	16#4417: sMsg := '4417 parameter „Tolerance window for modulo-start” The value for the tolerance window for the modulo-axis-start is invalid. The value must be greater or equal than zero and smaller than the half encoder modulo-perio…';
	16#4418: sMsg := '4418 parameter „Encoder reference mode” The value for the encoder reference mode is not allowed, resp. is not supported for this encoder type.';
	16#4419: sMsg := '4419 parameter „Encoder evaluation direction” The value for the encoder evaluation direction (log. counter direction) is not allowed.';
	16#441A: sMsg := '441A parameter „Encoder reference system” The value for the encoder reference system is invalid (0: incremental, 1: absolute, 2: absolute+modulo).';
	16#441B: sMsg := '441B parameter „Encoder position initialization mode” When starting the TC system the value for the encoder position initialization mode is invalid.';
	16#441C: sMsg := '441C parameter „Encoder sign interpretation (UNSIGNED- / SIGNED- data type)” The value for the encoder sign interpretation (data type) for the encoder the actual increment calculation (0: Default/not defined, 1: UNS…';
	16#4420: sMsg := '4420 parameter "Software end location monitoring minimum not allowed" The value for the activation of the software location monitoring minimum is not allowed.';
	16#4421: sMsg := '4421 parameter "Software end location monitoring maximum not allowed" The value for the activation of the software location monitoring maximum is not allowed.';
	16#4422: sMsg := '4422 function "Actual value setting is outside the value range" The "set actual value" function cannot be carried out, because the new actual position is outside the expected range of values.';
	16#4423: sMsg := '4423 parameter "Software end location minimum not allowed" The value for the software end location minimum is not allowed.';
	16#4424: sMsg := '4424 parameter "Software end location maximum not allowed" The value for the software end location maximum is not allowed.';
	16#4425: sMsg := '4425 parameter „Filter mask for the raw data of the encoder is invalid” The value for the filter mask of the encoder raw data in increments is invalid.';
	16#4426: sMsg := '4426 parameter „Reference mask for the raw data of the encoder is invalid” The value for the reference mask (increments per encoder turn, absolute resolution) for the raw data of the encoder is invalid. E.g. this va…';
	16#4430: sMsg := '4430 function "Hardware latch activation (encoder)" Activation of the encoder hardware latch was implicitly initiated by the referencing procedure. If this function has already been activated but a latch value has …';
	16#4431: sMsg := '4431 function "External hardware latch activation (encoder)" The activation of the external hardware latch (only available on the KL5101) is initiated explicitly by an ADS command (called from the PLC program of th…';
	16#4432: sMsg := '4432 function "External hardware latch activation (encoder)" If a referencing procedure has previously been initiated and the hardware still signals a valid latch value ("latch valid"), this function must not be ca…';
	16#4433: sMsg := '4433 function "External hardware latch activation (encoder)" If this function has already been initiated and the hardware is still signaling that the external latch value is still valid ("extern latch valid"), a fu…';
	16#4434: sMsg := '4434 monitoring "Encoder function not supported" An encoder function has been activated that is currently not released for use, or which is not even implemented.';
	16#4435: sMsg := '4435 monitoring „Encoder function is already active” An encoder function can not been activated because this functionality is already active.';
	16#4440: sMsg := '4440 initialization "Encoder initialization" Encoder has not been initialized. Although the axis has been created, the rest of the initialization has not been performed (1. Initialization of axis I/O, 2. Initialization o…';
	16#4441: sMsg := '4441 address "Axis address" The encoder does not have an axis, or the axis address has not been initialized.';
	16#4442: sMsg := '4442 address "I/O input structure address" The drive does not have a valid I/O input address in the process image.';
	16#4443: sMsg := '4443 address "I/O output structure address" The encoder does not have a valid I/O output address in the process image.';
	16#4450: sMsg := '4450 monitoring "Encoder counter underflow monitoring" The encoders incremental counter has underflowed.';
	16#4451: sMsg := '4451 monitoring "Encoder counter overflow monitoring" The encoders incremental counter has overflowed.';
	16#4460: sMsg := '4460 monitoring "Software end location minimum (axis start)" With active monitoring of the software end location for a minimum, a start has been made from a position that lies below the software end location minimum.…';
	16#4461: sMsg := '4461 monitoring "Software end location maximum (axis start)" With active monitoring of the software end location for a maximum, a start has been made from a position that lies above the software end location maximum.…';
	16#4462: sMsg := '4462 monitoring "Software end location minimum (positioning process)" With active monitoring of the software end location for a minimum, the actual position has fallen below the software end location minimum. In the …';
	16#4463: sMsg := '4463 monitoring "Software end location maximum (positioning process)" With active monitoring of the software end location for a maximum, the actual position has exceeded the software end location maximum. In the case…';
	16#4464: sMsg := '4464 monitoring „Encoder hardware error” The drive resp. the encoder system reports a hardware error of the encoder. An optimal error code is displayed in the message of the event log.';
	16#4465: sMsg := '4465 monitoring „Position initialization error at system start” At the first initialization of the set position was this for all initialization trials (without over-/under-flow, with underflow and overflow ) out of t…';
	16#4470: sMsg := '4470 monitoring "SSI transformation fault or not finished" The SSI transformation of the FOX 50 module was faulty for some NC-cycles or did not finished respectively.';
	16#44A2: sMsg := '44A2 monitoring "ENCERR_ADDR_CONTROLLER"';
	16#44A3: sMsg := '44A3 monitoring "ENCERR_INVALID_CONTROLLERTYPE"';
	16#4500: sMsg := '4500 parameter "Controller ID not allowed" The value for the controller ID is not allowed, e.g. because it has already been assigned, is less than or equal to zero, or is greater than 255.';
	16#4501: sMsg := '4501 parameter "Controller type not allowed" The value for the controller type is unacceptable because it is not defined. Type 1: P-controller (position) . . . Type 7: High/low speed controller Type 8: Stepper motor…';
	16#4502: sMsg := '4502 parameter "Controller operating mode not allowed" The value for the controller operating mode is not allowed.';
	16#4503: sMsg := '4503 parameter "Weighting of the velocity pre-control not allowed" The value for the percentage weighting of the velocity pre-control is not allowed. The parameter is pre-set to 1.0 (100%) as standard.';
	16#4504: sMsg := '4504 parameter "Following error monitoring (position) not allowed" The value for the activation of the following error monitoring is not allowed.';
	16#4505: sMsg := '4505 parameter "Following error (velocity) not allowed" The value for the activation of the following error monitoring (velocity) is not allowed.';
	16#4506: sMsg := '4506 parameter "Following error window (position) not allowed" The value for the following error window (maximum allowable following error) is not allowed.';
	16#4507: sMsg := '4507 parameter "Following error filter time (position) not allowed" The value for the following error filter time (position) is not allowed.';
	16#4508: sMsg := '4508 parameter "Following error window (velocity) not allowed" The value for the following error window (velocity) is not allowed.';
	16#4509: sMsg := '4509 parameter "Following error filter time (velocity) not allowed" The value for the following error filter time (velocity) is not allowed.';
	16#4510: sMsg := '4510 parameter "Proportional gain Kv or Kp (position controller) not allowed" The value for the proportional gain (Kv factor or Kp factor) is not allowed.';
	16#4511: sMsg := '4511 parameter "Integral-action time Tn (position controller) not allowed" The value for the integral-action time is not allowed (I proportion of the PID T1 controller).';
	16#4512: sMsg := '4512 parameter "Derivative action time Tv (position controller) not allowed" The value for the derivative action time is not allowed (D proportion of the PID T1 controller).';
	16#4513: sMsg := '4513 parameter "Damping time Td (position controller) not allowed" The value for the damping time is not allowed (D proportion of the PID T1 controller). Suggested value: 0.1 * Tv';
	16#4514: sMsg := '4514 function "Activation of the automatic offset compensation not allowed" Activation of the automatic offset compensation is only possible for certain types of controller (with no I component).';
	16#4515: sMsg := '4515 parameter "Additional proportional gain Kv or Kp (position controller) not allowed" The value for the second term of the proportional gain (Kv factor or Kp factor) is not allowed.';
	16#4516: sMsg := '4516 parameter "Reference velocity for additional proportional gain Kv or Kp (position controller) not allowed" The value for the reference velocity percentage data entry, to which the additional proportional gain i…';
	16#4517: sMsg := '4517 parameter "Proportional gain Pa (acceleration proportion) not allowed" The value for the proportional gain (Pa factor) is not allowed.';
	16#4518: sMsg := '4518 parameter "Proportional gain Kv (velocity controller) not allowed" The value for the proportional gain (Kv factor) is not allowed.';
	16#4519: sMsg := '4519 parameter “Reset time Tn (velocity controller) not allowed” The value for the integral-action time is not allowed (I proportion of the PID T1 controller).';
	16#451A: sMsg := '451A address "CONTROLERR_RANGE_ACCJUMPLIMITINGMODE"';
	16#451B: sMsg := '451B address "CONTROLERR_RANGE_ACCJUMPVALUE"';
	16#451C: sMsg := '451C address "CONTROLERR_RANGE_FILTERTIME"';
	16#451D: sMsg := '451D parameter „Dead zone not allowed” The value for the dead zone from the position error or the velocity error (system deviation) is not allowed (only for complex controller with velocity or torque interface).';
	16#4520: sMsg := '4520 parameter ”Rate time Tv (velocity controller) not allowed” The value for the derivative action time is not allowed (D proportion of the PID T1 controller).';
	16#4521: sMsg := '4521 parameter "Damping time Td (velocity controller) not allowed" The value for the damping time is not allowed (D proportion of the PID T1 controller). Suggested value: 0.1 * Tv';
	16#4522: sMsg := '4522 parameter "CONTROLERR_RANGE_IOUTPUTLIMIT"';
	16#4523: sMsg := '4523 parameter "CONTROLERR_RANGE_DOUTPUTLIMIT"';
	16#4524: sMsg := '4524 parameter "CONTROLERR_RANGE_POSIDISABLEWHENMOVING"';
	16#4540: sMsg := '4540 initialization "Controller initialisation" Controller has not been initialised. Although the controller has been created, the rest of the initialisation has not been performed (1. Initialisation of controller, 2. Re…';
	16#4541: sMsg := '4541 address "Axis address" Controller does not know its axis, or the axis address has not been initialised.';
	16#4542: sMsg := '4542 address "Drive address" Controller does not know its drive, or the drive address has not been initialised.';
	16#4550: sMsg := '4550 monitoring "Following error monitoring (position)" With active following error monitoring (position) a following error exceedance has occurred, whose magnitude is greater than the following error window, and who…';
	16#4551: sMsg := '4551 monitoring "Following error monitoring (velocity)" With active following error monitoring (velocity) a velocity following error exceedance has occurred, whose magnitude is greater than the following error window…';
	16#45A0: sMsg := '45A0 monitoring "CONTROLERR_RANGE_AREA_ASIDE"';
	16#45A1: sMsg := '45A1 monitoring "CONTROLERR_RANGE_AREA_BSIDE"';
	16#45A2: sMsg := '45A2 monitoring "CONTROLERR_RANGE_QNENN"';
	16#45A3: sMsg := '45A3 monitoring "CONTROLERR_RANGE_PNENN"';
	16#45A4: sMsg := '45A4 monitoring "CONTROLERR_RANGE_AXISIDPRESP0"';
	16#4600: sMsg := '4600 parameter "Drive ID not allowed" The value for the drive ID is not allowed, e.g. because it has already been assigned, is less than or equal to zero, or is greater than 255.';
	16#4601: sMsg := '4601 parameter "Drive type not allowed" The value for the drive type is unacceptable because it is not defined.';
	16#4602: sMsg := '4602 parameter "Drive operating mode not allowed" The value for the drive operating mode is not allowed. Modus 1: Standard';
	16#4603: sMsg := '4603 parameter "Motor polarity inverted?" The flag for the motor polarity is not allowed. Flag 0: Positive motor polarity Flag 1: Negative motor polarity';
	16#4604: sMsg := '4604 parameter "Drift compensation/velocity offset (DAC offset)" The value for the drift compensation (DAC offset) is not allowed.';
	16#4605: sMsg := '4605 parameter "Reference velocity (velocity pre-control)" The value for the reference velocity (velocity pre-control) is not allowed.';
	16#4606: sMsg := '4606 parameter "Reference output in percent" The value for the reference output in percent is not allowed. The value 1.0 (100 %) usually corresponds to a voltage of 10.0 V.';
	16#4607: sMsg := '4607 parameter "Quadrant compensation factor" The value for the quadrant compensation factor is not allowed.';
	16#4608: sMsg := '4608 parameter "Velocity reference point in percent" The value for the velocity reference point in percent is not allowed. The value 1.0 corresponds to 100 percent.';
	16#4609: sMsg := '4609 parameter "Output reference point in percent" The value for the output reference point in percent is not allowed. The value 1.0 corresponds to 100 percent.';
	16#460A: sMsg := '460A parameter "Minimum or maximum output limit" The values for the minimum and/or maximum output limit is not allowed. This will happen if the range of values is exceeded, the maximum limit is smaller than the mini…';
	16#460B: sMsg := '460B parameter "DRIVEERR_RANGE_MAXINCREMENT"';
	16#460C: sMsg := '460C parameter "DRIVEERR_RANGE_ DRIVECONTROLDWORD"';
	16#460D: sMsg := '460D parameter "DRIVEERR_RANGE_ RESETCYCLECOUNTER"';
	16#460F: sMsg := '460F parameter „Drive torque output scaling is not allowed” The value for the drive torque output scaling (rotary motor) or the force output scaling (linear motor) is not allowed.';
	16#4610: sMsg := '4610 parameter „Drive velocity output scaling is not allowed” The value for the drive velocity output scaling is not allowed.';
	16#4611: sMsg := '4611 parameter "Profi Drive DSC Proportional gain Kpc (position controller) not allowed" The value for the profi drive DSC proportional gain (Kpc factor) is not allowed.';
	16#4612: sMsg := '4612 parameter „Table-ID is invalid” The value for the table-ID is invalid.';
	16#4613: sMsg := '4613 parameter „Table interpolationtype is invalid” The value for the table interpolation-type is invalid.';
	16#4614: sMsg := '4614 parameter „Outputoffset in percent is invalid” The value for the output offset in percent (+/- 1.0) is invalid.';
	16#4615: sMsg := '4615 parameter „Profi Drive DSC scaling factor for calculating Xerr (position controller) is not allowed” The value as profi drive DSC scaling factor for calculating Xerr is invalid.';
	16#4616: sMsg := '4616 parameter „Drive acceleration output scaling is not allowed” The value for the drive acceleration/deceleration output scaling is not allowed.';
	16#4617: sMsg := '4617 parameter „Drive position output scaling is not allowed” The value for the drive position output scaling is not allowed.';
	16#4620: sMsg := '4620 parameter "Bit mask for stepper motor cycle not allowed" A value in the various stepper motor masks for the cycle concerned is not allowed.';
	16#4621: sMsg := '4621 parameter "Bit mask for stepper motor holding current not allowed" The value for the stepper motor holding mask is not allowed.';
	16#4630: sMsg := '4630 monitoring „Overtemperature” The drive resp. terminal detects an overtemperature alarm.';
	16#4631: sMsg := '4631 monitoring „Undervoltage” The drive resp. terminal detects an undervoltage (supply voltage to low).';
	16#4632: sMsg := '4632 monitoring „Wire breakage in phase A” The drive resp. terminal detects a wire breakage in phase A.';
	16#4633: sMsg := '4633 monitoring „Wire breakage in phase B” The drive resp. terminal detects a wire breakage in phase B.';
	16#4634: sMsg := '4634 monitoring „Overcurrent in phase A” The drive resp. terminal detects an overcurrent in phase A.';
	16#4635: sMsg := '4635 monitoring „Overcurrent in Phase B” The drive resp. terminal detects an overcurrent in phase B.';
	16#4636: sMsg := '4636 monitoring „Torque overload (stall situation)” The drive resp. terminal detects a torque overload (stall situation).';
	16#4640: sMsg := '4640 initialization "Drive initialisation" Drive has not been initialised. Although the drive has been created, the rest of the initialisation has not been performed (1. Initialisation of drive I/O, 2. Initialisation of …';
	16#4641: sMsg := '4641 address "Axis address" Drive does not know its axis, or the axis address has not been initialised.';
	16#4642: sMsg := '4642 address "I/O input structure address" The drive does not have a valid I/O input address in the process image.';
	16#4643: sMsg := '4643 address "I/O output structure address" The drive does not have a valid I/O output address in the process image.';
	16#4650: sMsg := '4650 monitoring "Drive not ready for operation" The drive is not ready for operation. The following are possible causes: - the drive is in failure state (hardware fault) - the drive is in the starting-up stage…';
	16#4651: sMsg := '4651 monitoring "Error in cyclic communication with the drive (life counter)"';
	16#4652: sMsg := '4652 monitoring "Not permitted to change the table ID while the axis is enabled"';
	16#4655: sMsg := '4655 monitoring "Invalid IO data for more than n consecutive nc cycles"';
	16#4A00: sMsg := '4A00 parameter "Table ID not allowed" The value for the table ID is not allowed, e.g. because it has already been assigned, is less than or equal to zero, or is greater than 255.';
	16#4A01: sMsg := '4A01 parameter "Table type not allowed" The value for the table type is unacceptable because it is not defined.';
	16#4A02: sMsg := '4A02 parameter "Number of lines in the table not allowed" The value of the number of lines in the table is not allowed, because, for example, it is smaller than two at linear interpolation and smaller than four at s…';
	16#4A03: sMsg := '4A03 parameter "Number of columns in the table is not allowed" The value of the number of columns in the table is not allowed, because, for example, it is less than or equal to zero (depends upon the type of table o…';
	16#4A04: sMsg := '4A04 parameter "Step size (position delta) not allowed" The value for the step size between two lines (position delta) is not allowed, because, for example, it is less than or equal to zero.';
	16#4A05: sMsg := '4A05 parameter "Period not allowed" The value for the period is not allowed, because, for example, it is less than or equal to zero.';
	16#4A06: sMsg := '4A06 parameter "Table is not monotonic" The value for the step size is not allowed, because, for example, it is less than or equal to zero.';
	16#4A07: sMsg := '4A07 initialization „Table sub type is not allowed” The value for the table sub type is not allowed or otherwise the table class (slave type) do not match up to the table main type.';
	16#4A08: sMsg := '4A08 initialization „Table interpolation type is not allowed” The value for the table interpolation type is allowed.';
	16#4A09: sMsg := '4A09 initialization "Incorrect table main type" The table main type is unknown or otherwise the table class (slave type) do not match up to the table main type.';
	16#4A10: sMsg := '4A10 initialization "Table initialisation" Table has not been initialised. Although the table has been created, the rest of the initialisation has not been performed. For instance, the number of lines or columns may be l…';
	16#4A11: sMsg := '4A11 initialization "Not enough memory" Table could not be created, since there is not enough memory.';
	16#4A12: sMsg := '4A12 function "Function not executed, function not available" The function has not been implemented, or cannot be executed, for the present type of table.';
	16#4A13: sMsg := '4A13 function "Line index not allowed" The start line index or the stop line index to be used for read or write access to the table is not allowed. For instance, the line index may be greater than the total number …';
	16#4A14: sMsg := '4A14 function "Column index not allowed" The start column index or the stop column index to be used for read or write access to the table in not allowed. For instance, the column index may be greater than the total…';
	16#4A15: sMsg := '4A15 function "Number of lines not allowed" The number of lines to be read from or written to the table is not allowed. The number of lines must be an integer multiple of the number of elements in a line (n * numbe…';
	16#4A16: sMsg := '4A16 function "Number of columns not allowed" The number of columns to be read from or written to the table is not allowed. The number of columns must be an integer multiple of the number of elements in a column (n…';
	16#4A17: sMsg := '4A17 function "Error in scaling or in range entry" The entries in the table header are inconsistent, e.g. the validity range is empty. If the error is generated during the run time it is a run time error and stops …';
	16#4A18: sMsg := '4A18 function "Multi table slave out of range" The slave master position is outside the table values for the master. The error is a run-time error, and stops the master/slave group.';
	16#4A19: sMsg := '4A19 function "Solo table underflow" The slave master position is outside the table values for the master. The master value of the equidistant table, to be processed linearly, lies under the first table value. The …';
	16#4A1A: sMsg := '4A1A function "Solo table overflow" The slave master position is outside the table values for the master. The master value of the equidistant table, to be processed linearly, lies above the first table value. The e…';
	16#4A1B: sMsg := '4A1B parameter "Incorrect execution mode" The cyclic execution mode can only be "true" or "false".';
	16#4A1C: sMsg := '4A1C parameter "Impermissible parameter" The Fifo parameter is not allowed.';
	16#4A1D: sMsg := '4A1D parameter "Fifo is empty" The Fifo of the external generator is empty. This can signify end of track or a run time error.';
	16#4A1E: sMsg := '4A1E parameter "Fifo is full" The Fifo of the external generator is full. It is the user‘s task to continue to attempt to fill the Fifo with the rejected values.';
	16#4A1F: sMsg := '4A1F parameter „Point-Index of Motion Function invalid” The point index of a Motion Function Point of a Function Table is invalid. First the point index has to be larger than zero and second it has to be numerical c…';
	16#4A20: sMsg := '4A20 initialization „No diagonalisation of matrix” The spline can not be calculated. The master positions are not correct.';
	16#4A21: sMsg := '4A21 initialization „Number of spline points to less” The number of points of a cubic spline has to be greater than two.';
	16#4A22: sMsg := '4A22 initialization „Fifo must not be overwritten” Fifo must not be overwritten since then the active line would be overwritten. It is the task of the user to secure that the active line is not modified.';
	16#4B00: sMsg := '4B00 parameter "Axis has been stopped" The axis has been stopped while the axis moves to target position. The axis could be stopped with a PLC Command via ADS, with the call of AXFNC or with the TwinCAT System Manag…';
	16#4B01: sMsg := '4B01 parameter "Axis cannot be started" The axis cannot be started, because:';
	16#4B02: sMsg := '4B02 parameter "Control mode not allowed" No Target Position Control and no Position Area Control.';
	16#4B03: sMsg := '4B03 parameter "Axis is not moving" Restart position and velocity is only allowed if axis is physically moving.';
	16#4B04: sMsg := '4B04 parameter "Wrong mode for RestartPosAndVelo" Wrong mode.';
	16#4B05: sMsg := '4B05 parameter "Command not allowed"';
	16#4B06: sMsg := '4B06 parameter "Parameter not correct"';
	16#4B07: sMsg := '4B07 parameter "Timeout axis function block"';
	16#4B08: sMsg := '4B08 parameter "Axis in protected mode" Axis is in protected mode (i.e. coupled) and cannot be moved.';
	16#4B09: sMsg := '4B09 parameter "Axis is not ready" Axis is not ready and cannot be moved.';
	16#4B0A: sMsg := '4B0A parameter "Homing error" The Homing of an axis could not be started or was not successful';
	16#4B0B: sMsg := '4B0B parameter "Invalid definition trigger input definition" The definition of the trigger signal used with the function block MC_TouchProbe is invalid. The defined encoder ID, the trigger signal or the trigger sign…';
	16#4B0C: sMsg := '4B0C function "position latch has been deactivated" The function block MC_TouchProbe encountered that a touch probe sequence has been deactivated after the block started this sequence. The reason for instance can b…';
	16#4B0D: sMsg := '4B0D function "Timeout NC status feedback" A function block has successfully executed a command but the NC does not pass the expected feedback in the axis status word.';
	16#4B0E: sMsg := '4B0E function "Supplement not installed" - The function is available as supplement product but not installed on the system.';
	16#4B0F: sMsg := '4B0F function "Timeout Register Access" - The access to a bus terminal register timed out.';
	16#4B10: sMsg := '4B10 function "M-Function request missing" This error occurs if a confirmation of an M-Function is made but the request bit is not set.';
	16#4B11: sMsg := '4B11 parameter "Zero shift index is out of range" The index of the zero shift is invalid';
	16#4B12: sMsg := '4B12 parameter "R parameter index or size is invalid". This error occurs, if the R parameters are written or read and the index or size is out of range';
	16#4B13: sMsg := '4B13 parameter "Index for tool description is invalid"';
	16#4B14: sMsg := '4B14 function "Version of cyclic channel interface does not match to the requested function and function block, resp." This error occurs, if an older TwinCAT Version is used and a new functionality from a newer TcN…';
	16#4B15: sMsg := '4B15 function "Channel is not ready for requested function". The requested function can not be executed due to a wrong state of the channel. This error occurs for instance, if retrace is requested and the axes are …';
	16#4B16: sMsg := '4B16 function "Requested function is not turned on". The requested function requires an explicit activation before it can be executed.';
	16#4B20: sMsg := '4B20 parameter "Cannot append all axes". This error occurs, if you want to append an auxiliary axes to an interpolation group and the function fails. Probably a prior assignment of an auxiliary axes was skipped.';
	16#4B30: sMsg := '4B30 parameter "Pointer invalid". The pointer to a data structure is invalid, e.g. NULL.';
	16#4B31: sMsg := '4B31 parameter "Size of memory invalid". The size parameter is invalid.';
	16#4B32: sMsg := '4B32 parameter "Invalid cam table ID". The cam table ID is out of the range from 1 to 255.';
	16#4B33: sMsg := '4B33 parameter "Invalid point ID". The point ID of a motion function point is lower than 1.';
	16#4B34: sMsg := '4B34 parameter "Invalid number of points ". The number of points to read or write is less than 1.';
	16#4B35: sMsg := '4B35 parameter "Invalid MC table type". The type of a cam table does not match the MC_TableType definition.';
	16#4B36: sMsg := '4B36 parameter "Invalid number of rows". The number of rows of a cam table is less than 1.';
	16#4B37: sMsg := '4B37 parameter "Invalid number of columns". The number of columns of a cam table is invalid.';
	16#4B38: sMsg := '4B38 parameter "Invalid Increment". The increment for an interpolation is invalid, e.g. <= 0.';
	16#4B40: sMsg := '4B40 monitoring "Unsupported Terminal Type". The terminal in use is not supported by this function block.';
	16#4B41: sMsg := '4B41 monitoring "Register Read/Write Error". This error implies to be a validation error.';
	16#4B42: sMsg := '4B42 monitoring "Axis is Enabled". Axis is enabled and is not supposed to be enabled for this operation';
	16#4B43: sMsg := '4B43 parameter "Size of compensation table wrong". The stated table size in bytes is not conform with the real size.';
	16#4B44: sMsg := '4B44 parameter The minimum/ maximum position of the compenstation table is not conform to the position in the table description (ST_CompensationDesc)';
	16#4B45: sMsg := '4B45 parameter "Not implemented". The requested function is not implemented in this combination.';
	16#4B60: sMsg := '4B60 monitoring "Motion command not be activated". A motion command has been started and has been buffered and confirmed by the NC. Nevertheless the command did not become active.';
	16#4B61: sMsg := '4B61 monitoring "Motion command could not be monitored by the PLC". A motion command has been started and has been buffered and confirmed by the NC. The PLC has not been able to monitor the execution of this command……';
	16#4B62: sMsg := '4B62 monitoring "Buffered command finished with error". A buffered command finished with an error. The error number is not available because a new command is already in execution.';
	16#4B63: sMsg := '4B63 monitoring "Buffered command finished without state feedback". A buffered command finished without success or error feedback.';
	16#4B64: sMsg := '4B64 monitoring "  BufferMode  not supported". The  BufferMode  is not supported by the command.';
	16#4B65: sMsg := '4B65 monitoring "Command number is zero". The system administrated command number for buffered commands is zero. ';
	16#4B71: sMsg := '4B71 parameter "Invalid NCI Entry Type". FB_NciFeedTablePreparation is called with an unknown nEntryType';
	16#4B72: sMsg := '4B72 function "NciFeedTable full". The table is full filled and therefore this entry is not accepted.';
	16#4B73: sMsg := '4B73 function internal error';
	16#4B74: sMsg := '4B74 parameter "ST_NciTangentialFollowingDesc: tangential axis is not an auxiliary axis" The entry ST_NciTangentialFollowingDesc contains an tangential axis that is no auxiliary axis.';
	16#4B75: sMsg := '4B75 parameter ST_NciTangentialFollowingDesc: nPathAxis1 and nPathAxis2, resp. are no path axes. So it is not possible to determine the plane.';
	16#4B76: sMsg := '4B76 parameter ST_NciTangentialFollwoingDesc: nPathAxis1 and nPathAxis2 are equal. So it is not possible to determine the plane.';
	16#4B77: sMsg := '4B77 parameter ST_NciGeoCirclePlane: circle is programmed in a wrong manner.';
	16#4B78: sMsg := '4B78 function Internal error in calculation of the tangential following';
	16#4B79: sMsg := '4B79 monitoring Tangential following: With ST_NciTangentialFollowingDesc the monitoring of the deviation angle (E_TfErrorOnCrirical1) is activated and with the actual segment the deviation angle is too big.';
	16#4B7A: sMsg := '4B7A function not implemented';
	16#4B7B: sMsg := '4B7B parameter Tangential Following: The radius of the actual circle segment is too small';
	16#4B7C: sMsg := '4B7C parameter FB_NciFeedTablePreparation: pEntry is NULL';
	16#4B7D: sMsg := '4B7D parameter FB_NciFeedTablePreparation: The specified nEntryType does not match the the structure type';
	16#4B7E: sMsg := '4B7E parameter ST_NciMFuncFast and ST_NciMFuncHsk: The requested m-function is not in between 0..159';
	16#4B7F: sMsg := '4B7F parameter ST_NciDynOvr: The requested value for the dynamic override is not in between 0.01 and 1.0';
	16#4B80: sMsg := '4B80 parameter ST_NciVertexSmoothing: invalid parameter. This error occurs with a negative vertex radius or an unknown vertex smoothing type.';
	16#4B81: sMsg := '4B81 parameter FB_NciFeedTablePrepartion: The requested velocity is not in a valid range';
	16#4B82: sMsg := '4B82 parameter ST_Nci*: invalid parameter';

ELSE
	sMsg := UDINT_TO_STRING(iErrID);
	sMsg := concat(sMsg, ' Unknown Error code');
END_CASE
F_AxErrMsg := sMsg;

END_FUNCTION

// ---- AxisOnline/FB_McAxisOnline_EL72xx.TcPOU
//==================================================================================================
//							Beckhoff Automation Poland
//									06.02.2024
//	Basic Axis Function Block object to control mostly used functionabilities, 
//	Required libs: Tc2_EtherCAT, Tc2_MC2_Drive, Tc2_MC2
// 	v2.0	|| TC v 3.1.4024.53		|| New release. Inheritance added.
//  v1.1	|| TC v 3.1.4022.27		|| ACT_SetPositionIO - Changed FB type to FB_CoeEL72xxSetPositionOffset
// 	v1.0 	|| TC v 3.1.4022.22	 	|| First release
//==================================================================================================
{attribute 'reflection'}
FUNCTION_BLOCK FB_McAxisOnline_EL72xx EXTENDS FB_McAxisOnline_NC
VAR_INPUT
END_VAR
VAR_OUTPUT
END_VAR
VAR
	fbMotorMonitoring					: FB_MotorMonitoringEL72xx;
	fbHoldingBrakeCtrl					: FB_HoldingBrakeCtrlEL72xx;
	tonGetDriveDiag						: TON;
	fbReadChannelErrorCode				: FB_ReadChannelErrorCodeEL72xx;
	fbSetPositionOffset					: FB_CoeEL72xxSetPositionOffset;	// Requires FW >= 19 Rev >= 30!		(check motor type if have multiturn enc to save in enc)		https://infosys.beckhoff.com/content/1033/tcplclib_tc2_mc2_drive/7604235915.html?id=9112637119101863462
	fbDeletePositionOffset				: FB_CoEEL72xxDeletePositionOffset;
	mcReadDriveAddress					: MC_ReadDriveAddress;
	fbGetDriveRef						: FB_GetDriveRef;
	
	// Initialization
	bDriveAddressReady					: BOOL;
	bDriveRefReady						: BOOL;
END_VAR

// Device dependent initialization 
M_Init_EL72xx();
// Device independent commands, mostly NC 
M_States();
M_SWLimitSwitch();
M_Stop();
M_Power();
M_Homing();
M_Jog();
M_Move();
M_Reset();
M_SetPosition();
// Device dependent commands
// Motor monitoring possible only with real axis
IF NOT AxisRef.Status.OpMode.SimulationAxis THEN
	M_MotorMonitoring();
END_IF
// Device dependent commands, possible only on real axis after complete initialization
IF bInitialized AND NOT AxisRef.Status.OpMode.SimulationAxis THEN
	M_SetPositionIO();
	M_DeletePositionIO();
	M_DriveDiag();
	M_HoldingBrakeCtrl();
END_IF

// Device independent error collection
M_ErrorCollection();

METHOD M_DeletePositionIO : BOOL
VAR_INPUT
END_VAR
// Requires module FW >= 19 Rev >= 30!		
// Requires library: Tc2_MC2_Drive ≥ V3.3.17.0
// Check motor type if have multiturn enc to save in enc. (Motor with singleturn feedback and eMemory.Encoder = error without execute = 0x4BB4)
// https://infosys.beckhoff.com/content/1033/tcplclib_tc2_mc2_drive/7604235915.html?id=9112637119101863462
	
fbDeletePositionOffset(
	Axis		:= AxisRef, 
	Execute		:= Axis.stDeletePositionOffset.bExecute, 
	Feedback	:= Axis.stDeletePositionOffset.eFeedback, 
	Memory		:= Axis.stDeletePositionOffset.eMemory, 
	Busy		=> Axis.stDeletePositionOffset.bBusy, 
	Error		=> Axis.stDeletePositionOffset.bError, 
	ErrorID		=> Axis.stDeletePositionOffset.udiErrorID);
END_METHOD

METHOD M_DriveDiag : BOOL
VAR_INPUT
END_VAR
// Auto update when drive error
tonGetDriveDiag(	IN	:= Axis.stError.bDriveError AND NOT tonGetDriveDiag.Q, 
					PT	:= T#5S, 
					Q	=> , 
					ET	=> );

fbReadChannelErrorCode(	bExecute				:= Axis.stChannelErrorCode.bExecute OR tonGetDriveDiag.Q,
						stDriveRef				:= Axis.stDriveRef,
						bBusy					=> Axis.stChannelErrorCode.bBusy,
						bError					=> Axis.stChannelErrorCode.bError,
						uiAdsErrId				=> Axis.stChannelErrorCode.uiAdsErrId,
						uiCANopenErrId			=> Axis.stChannelErrorCode.uiSecErrId,
						uiChannelErrorCode		=> Axis.stChannelErrorCode.uiChannelErrorCode,
						uiChannelErrorCodeHex	=> Axis.stChannelErrorCode.uiChannelErrorCodeHex);
END_METHOD

METHOD M_ErrorCollection : BOOL
VAR_INPUT
END_VAR
// Error flags
Axis.stError.bDriveError					:= AxisRef.Status.DriveDeviceError;

Axis.stError.bNcError						:= AxisRef.Status.Error;

Axis.stError.bFBError						:= Axis.mcPower.bError OR Axis.mcReset.bError OR Axis.mcHome.bError OR Axis.mcJog.bError
													OR Axis.mcHalt.bError OR Axis.mcStop.bError OR Axis.mcSS1.bError OR Axis.mcSS2.bError
													OR Axis.mcMoveAbsolute.bError OR Axis.mcMoveRelative.bError OR Axis.mcMoveVelocity.bError OR Axis.mcMoveModulo.bError
													OR Axis.mcMoveAbsolute2.bError OR Axis.mcMoveRelative2.bError OR Axis.mcMoveVelocity2.bError OR Axis.mcMoveModulo2.bError
													OR Axis.stNcLimitSwitch.bError OR Axis.mcSetPosition.bError;
									
Axis.stError.bCommunicationError			:= Axis.stChannelErrorCode.bError OR Axis.stSetPositionOffset.bError OR Axis.stMotorMonitoring.bError OR Axis.stHoldingBrake.bError;

Axis.stError.bError						:= Axis.stError.bDriveError OR Axis.stError.bNcError OR Axis.stError.bFBError OR Axis.stError.bCommunicationError;
Axis.bError								:= Axis.stError.bError; // Forward one stage up

// Error codes
Axis.stError.uiDriveErrorID 				:= Axis.stChannelErrorCode.uiChannelErrorCode;
Axis.stError.uiDriveErrorIDHex 			:= Axis.stChannelErrorCode.uiChannelErrorCodeHex;

Axis.stError.udiNcErrorID 				:= AxisRef.Status.ErrorID;
Axis.stError.udiNcErrorIDHex 				:= AxisRef.Status.ErrorID;
	

Axis.stError.udiFBErrorID 				:= 	Axis.mcPower.udiErrorID + 
														Axis.mcReset.udiErrorID + 
														Axis.mcHome.udiErrorID + 
														Axis.mcJog.udiErrorID +
														Axis.mcHalt.udiErrorID + 
														Axis.mcStop.udiErrorID + 
														Axis.mcSS1.udiErrorID + 
														Axis.mcSS2.udiErrorID +
														Axis.mcMoveAbsolute.udiErrorID + 
														Axis.mcMoveRelative.udiErrorID + 
														Axis.mcMoveVelocity.udiErrorID + 
														Axis.mcMoveModulo.udiErrorID +
														Axis.mcMoveAbsolute2.udiErrorID + 
														Axis.mcMoveRelative2.udiErrorID + 
														Axis.mcMoveVelocity2.udiErrorID + 
														Axis.mcMoveModulo2.udiErrorID +
														Axis.stNcLimitSwitch.udiErrorID + 
														Axis.mcSetPosition.udiErrorID;

Axis.stError.udiFBErrorIDHex 				:= Axis.stError.udiFBErrorID;

Axis.stError.udiErrorID					:= Axis.stSetPositionOffset.udiErrorID;
Axis.stError.uiAdsErrorID					:= Axis.stChannelErrorCode.uiAdsErrId + Axis.stMotorMonitoring.uiAdsErrId + Axis.stHoldingBrake.uiAdsErrId;
Axis.stError.uiSecErrorID					:= Axis.stChannelErrorCode.uiSecErrId + Axis.stMotorMonitoring.uiSecErrId + Axis.stHoldingBrake.uiSecErrId;

Axis.stError.sNcError						:= F_AxErrMsg(Axis.stError.udiNcErrorID);
Axis.stError.sDriveError					:= F_EL72ErrMsg(Axis.stError.uiDriveErrorID);
END_METHOD

METHOD M_HoldingBrakeCtrl : BOOL
VAR_INPUT
END_VAR
fbHoldingBrakeCtrl(bForceUnlock			:= Axis.stHoldingBrake.bForceUnlock,
					stDriveRef			:= Axis.stDriveRef,
					bBusy				=> Axis.stHoldingBrake.bBusy,
					bError				=> Axis.stHoldingBrake.bError,
					uiAdsErrId			=> Axis.stHoldingBrake.uiAdsErrId,
					uiCANopenErrId		=> Axis.stHoldingBrake.uiSecErrId);
END_METHOD

METHOD M_Init_EL72xx : BOOL
VAR_INPUT
END_VAR
// bInitialized flag is set just once. 
// bReInitialized ise set each time we do online change or request reinit operation
// bDriveAddressReady, bReadParameterSetReady, bDriveRefReady - set just once after successed read

// Online change detection
bOnlineChangeDetected					:= udiOnlineChangeCntOld <> TwinCAT_SystemInfoVarList._AppInfo.OnlineChangeCnt;
udiOnlineChangeCntOld 					:= TwinCAT_SystemInfoVarList._AppInfo.OnlineChangeCnt;
// Reset init
IF bReInit OR bOnlineChangeDetected THEN
	iInitStep							:= 0;
END_IF

//Initialization process
CASE iInitStep OF
	0:	// Read Drive Address
		
		Axis.mcReadDriveAddress.bExecute	:=	 TRUE;
		iInitStep						:= iInitStep + 10;
		
	10: // Wait for data
	
		IF NOT Axis.mcReadDriveAddress.bBusy THEN
			Axis.mcReadDriveAddress.bExecute	:=	 FALSE;
			IF Axis.mcReadDriveAddress.bDone THEN
				iInitStep 				:= iInitStep + 10;
				bDriveAddressReady 		:= TRUE;
			ELSE
				iInitStep 				:= 1000;		// Error step
			END_IF
		END_IF
		
	20:	// Read Parameter Set
		
		Axis.mcReadParameterSet.bExecute		:=	 TRUE;
		iInitStep						:= iInitStep + 10;
		
	30: // Wait for data
	
		IF NOT Axis.mcReadParameterSet.bBusy THEN
			Axis.mcReadParameterSet.bExecute	:=	 FALSE;
			IF Axis.mcReadParameterSet.bDone THEN
				iInitStep 				:= iInitStep + 10;
				bReadParameterSetReady 	:= TRUE;
			ELSE
				iInitStep 				:= 1000;		// Error step
			END_IF
		END_IF	
	
	40:	// Get Drive Ref
		
		Axis.stGetDriveRef.bExecute		:=	 TRUE;
		iInitStep						:= iInitStep + 10;
		
	50: // Wait for data
	
		IF NOT Axis.stGetDriveRef.bBusy THEN
			Axis.stGetDriveRef.bExecute	:=	 FALSE;
			IF NOT Axis.stGetDriveRef.bError THEN
				iInitStep 				:= iInitStep + 10;
				bDriveRefReady 			:= TRUE;
			ELSE
				iInitStep 				:= 1000;		// Error step
			END_IF
		END_IF
	
	60: // Success - initialized flag, clear error
		bReInitialized					:= bInitialized;	// TRUE only when it's not first initialization e.g. online change
		bInitialized 					:= TRUE;
		bReInitializationError			:= FALSE;			// TRUE only when it's not first initialization e.g. online change
		bInitializationError			:= FALSE;
		iInitStep 						:= iInitStep + 10;
		
	70: // Idle
	
		;
		
	1000: // Error step
		wInitializationErrorCounter 	:= wInitializationErrorCounter + 1;
		IF wInitializationErrorCounter < 100 THEN
			iInitStep					:= iInitStep + 5;			// Go to delay
		ELSE
			bReInitializationError		:= bInitializationError;	// TRUE only when it's not first initialization e.g. online change
			bInitializationError		:= TRUE;
			bReInitialized				:= FALSE;
			iInitStep 					:= iInitStep + 10;
		END_IF

	1005: // Delay step
		tonDelay(IN:= TRUE, PT:= T#1S);
		IF tonDelay.Q THEN
			tonDelay(IN:= FALSE, PT:= T#1S);
			iInitStep					:= 0;
		END_IF
		
	1010: // Idle after error
		;
	
END_CASE

mcReadDriveAddress(	Axis				:= AxisRef,
					Execute				:= Axis.mcReadDriveAddress.bExecute,
					Done				=> Axis.mcReadDriveAddress.bDone,
					Busy				=> Axis.mcReadDriveAddress.bBusy,
					Error				=> Axis.mcReadDriveAddress.bError,
					ErrorID				=> Axis.mcReadDriveAddress.udiErrorID,
					DriveAddress		=> Axis.stDriveAddress);
				
mcReadParameterSet(	Parameter			:= Axis.stAxisParameter,
					Axis				:= AxisRef,
					Execute				:= Axis.mcReadParameterSet.bExecute,
					Done				=> Axis.mcReadParameterSet.bDone,
					Busy				=> Axis.mcReadParameterSet.bBusy,
					Error				=> Axis.mcReadParameterSet.bError,
					ErrorID				=> Axis.mcReadParameterSet.udiErrorID);
					
fbGetDriveRef(		bExecute			:= Axis.stGetDriveRef.bExecute,
					bBusy				=> Axis.stGetDriveRef.bBusy,
					bError				=> Axis.stGetDriveRef.bError,
					udiErrorID			=> Axis.stGetDriveRef.udiErrorID,
					stDriveRef			=> Axis.stDriveRef,
					Axis				:= AxisRef);
END_METHOD

METHOD M_MotorMonitoring : BOOL
VAR_INPUT
END_VAR
fbMotorMonitoring(	bReset				:= Axis.stMotorMonitoring.bReset,
					rTorqueLimit		:= Axis.stMotorMonitoring.rTorqueLimit,
					stDriveRef			:= Axis.stDriveRef,
					bError				=> Axis.stMotorMonitoring.bError,
					uiAdsErrId			=> Axis.stMotorMonitoring.uiAdsErrId,
					uiCANopenErrId		=> Axis.stMotorMonitoring.uiSecErrId,
					bInitialized		=> Axis.stMotorMonitoring.bInitialized,
					bWarning			=> Axis.stMotorMonitoring.bWarning,
					rWarningCurrent		=> Axis.stMotorMonitoring.rWarningCurrent,
					rTorquePerc			=> Axis.stMotorMonitoring.rTorquePerc,
					rTorquePercMax		=> Axis.stMotorMonitoring.rTorquePercMax,
					rTorque				=> Axis.stMotorMonitoring.rTorque,
					rTorqueF			=> Axis.stMotorMonitoring.rTorqueF,
					rTorqueMax			=> Axis.stMotorMonitoring.rTorqueMax,
					rCurrent			=> Axis.stMotorMonitoring.rCurrent,
					rCurrentF			=> Axis.stMotorMonitoring.rCurrentF,
					rCurrentMax			=> Axis.stMotorMonitoring.rCurrentMax,
					rI2T				=> Axis.stMotorMonitoring.rI2T,
					rI2TMax				=> Axis.stMotorMonitoring.rI2TMax,
					Axis				:= AxisRef);
END_METHOD

METHOD M_SetPositionIO : BOOL
VAR_INPUT
END_VAR
// Requires module FW >= 19 Rev >= 30!		
// Requires library: Tc2_MC2_Drive ≥ V3.3.17.0
// Check motor type if have multiturn enc to save in enc. (Motor with singleturn feedback and eMemory.Encoder = error without execute = 0x4BB4)
// https://infosys.beckhoff.com/content/1033/tcplclib_tc2_mc2_drive/7604235915.html?id=9112637119101863462

fbSetPositionOffset(
	Axis		:= AxisRef, 
	Execute		:= Axis.stSetPositionOffset.bExecute,
	Position	:= Axis.stSetPositionOffset.lrPosition,
	Relative	:= Axis.stSetPositionOffset.bRelative, 
	Feedback	:= Axis.stSetPositionOffset.eFeedback, 
	Memory		:= Axis.stSetPositionOffset.eMemory,   
	Busy		=> Axis.stSetPositionOffset.bBusy,     
	Error		=> Axis.stSetPositionOffset.bError,    
	ErrorID		=> Axis.stSetPositionOffset.udiErrorID	);
END_METHOD

END_FUNCTION_BLOCK

// ---- AxisOnline/POUs/EL72xx/FB_MotorMonitoringEL72xx.TcPOU
//==================================================================================================
//							Beckhoff Automation Poland
//									21.03.2022
//	Blok funkcyjny pozwala na monitorowanie i ograniczanie momentu oraz monitoring parametru I2T dla EL72xx.
//	Zmienne do zlinkowania zadeklarowane są wewnątrz bloku.
//	Ograniczenie i monitorowanie momentu
//	Ograniczenie momentu podawane jest przez wejście rTorqueLimit.
//	Na wyjściu podana jest wartość surowa w %, jak i przeskalowana na A (prąd) i Nm (moment).
//	Blok zwraca wartości bieżące, przefiltrowane i maksymalne.
//	Wartości maksymalne mogą być wyzerowane za pomocą zmiennej bReset.
//	Wewnętrznie wykorzystany jest blok FB_FilterEx.
//
//	v1.1	|| TC v 3.1.4024.25		|| - Zaktualizowane skalowanie rTorqueF
//  v1.0	|| TC v 3.1.4022.22		|| - pierwsza wersja
//==================================================================================================
FUNCTION_BLOCK FB_MotorMonitoringEL72xx
VAR CONSTANT
	rTorqueLimitLow					: REAL 		:= 0.01;				// Low limit used for bipolar torque limit value
	rTorqueLimitHigh				: REAL		:= 500.0;				// High limit used for bipolar torque limit value
END_VAR
VAR_INPUT
	bReset							: BOOL;								// Reset FB
	rTorqueLimit					: REAL 		:= rTorqueLimitHigh; 	// Bipolar torque limit: 0-500%, resolution 0.1%, value goes to: 16#6072 (Ch A)/ 16#6872 (Ch B)	
	stDriveRef						: ST_DriveRef;						// Necessary for FB_CoERead_ByDriveRef
END_VAR
VAR_OUTPUT
	bError							: BOOL; 							// General error: parameter or CoE read.
																		// If bError = TRUE and bInitialized = FALSE - error during read motor data.
																		// If bError = TRUE and bInitialized = TRUE and (iAdsErrId <> 0 or iCANopenErrId <> 0) then I2T read error
																		// If bError = TRUE and bInitialized = TRUE and iAdsErrId = 0 and iCANopenErrId = 0 then parameter error: rTorqueLimit outside permitted range rTorqueLimitLow..rTorqueLimitHigh or Empty stDriveRef
	uiAdsErrId						: UINT;								// Forwarded output FB_CoERead_ByDriveRef
	uiCANopenErrId					: UINT;								// Forwarded output FB_CoERead_ByDriveRef
	bInitialized					: BOOL;								// TRUE - Motor data read without errors, so it's possible to calculate torqe and current values in metric units
	bWarning						: BOOL;								// rCurrentF > rWarningCurrent, be aware to be over permitted range
	rWarningCurrent					: REAL; 							// 8011:12 - Rated current in [A]
	rTorquePerc						: REAL;								// [%]
	rTorquePercMax					: REAL;								// Max [%]
	rTorque							: REAL; 							// [Nm]
	rTorqueF						: REAL;								// Filtered [Nm]
	rTorqueMax						: REAL;								// Max [Nm]
	rCurrent						: REAL; 							// [A]
	rCurrentF						: REAL;								// Filtered [A]
	rCurrentMax						: REAL;								// Max [A]
	rI2T							: REAL; 							// Thermal Motor Utilization: 16#32C1:02 (Ch A)/ 16#36C1:02 (Ch B); units: [%]
	rI2TMax							: REAL; 							// Max % Nominal
END_VAR
VAR_IN_OUT
	Axis							: AXIS_REF;							// Axis Ref struct
END_VAR
VAR
//======================= Internal var ===========================
	iStep							: INT;								// Case instruction
	bDriveRefOK						: BOOL;								// stDriveRef contains necessary data to read CoE
	bTorqueLimitOK					: BOOL;								// rTorqueLimit in permitted range rTorqueLimitLow..rTorqueLimitHigh
	uiBipolarTorqueLimitValue  		AT %Q*: UINT; 						// Raw data, linked to Bipolar torque limit value
	rTorqueRAW						: REAL; 							// -1000 .. 1000 - RAW values the same as process image
	rSfTorque						: REAL; 							// A --> Nm
	rSfCurrent						: REAL; 							// RAW -1000..1000 --> A
	wInitErrorCount					: WORD;								// Initialization error counter, if bigger then 10 then error
	rPeakCurrent					: REAL; 							// 8011:11 in [A]
	rRatedCurrent					: REAL; 							// 8011:12 in [A]
	bFirstCycle						: BOOL := TRUE;
	bRMSValue						: BOOL;								// 16#8010:54  Bit 0 = 1 - RMS value
//========================== EL72xx =============================
	dwPeakCurrent					: DWORD;							// 16#8011:11 - Max current, Peak current [mA]
	dwRatedCurrent					: DWORD;							// 16#8011:12 - Rated current [mA]
	dwTorqueConstant				: DWORD;							// 16#8011:16 - Torque constant [mNm/A]
	dwFeatureBits					: DWORD;							// 16#8010:54 - Feature bits:	Peak value --> Bit 0 = 0 (default for EL7201-000x) 
																									//	RMS value --> Bit 0 = 1 (default for EL7211-000x)
//========================== I2T ================================
	sDeviceName						: STRING;							// 
	sNo								: STRING(1);						// xxxxxxx-000Y - char Y
	usiI2T							: USINT;							// 
	bDS402Profile					: BOOL;								// Flag DS402
	bMDP742Profile					: BOOL;								// Flag MDP742
	wMotorI2TIndex					: WORD;								// EL72x1-0000 --> MDP 742: A011:11 Motor I2T temperature [%] USINT
																		// EL72x1-0001 --> DS 402: 2031:11 Motor I2T temperature [%] USINT
//========================== FBs ================================
	rtReset							: R_TRIG;							// Reset trigger
	tonWait							: TON;								// Wait timer
	fbFilterEx						: FB_FilterEx;						// Filter
	fbGETCURTASKINDEX   			: GETCURTASKINDEX;					// FB to check task no
	fbCoERead						: FB_CoERead_ByDriveRef;			// FB for read CoE parameters
//===============================================================
END_VAR

//===== Initialization, reinitialization and reset  =============
ACT_Init_Reset();
//=================== Call triggers and timers ==================
tonWait(IN:= NOT tonWait.Q, PT:= T#1S);
//======= Check for parameter error - each cycle ================
bDriveRefOK 							:= (stDriveRef.nSlaveAddr <> 0) AND (stDriveRef.sNetId <> '');
bTorqueLimitOK 							:= (rTorqueLimit > rTorqueLimitLow);
//============= Read params and calculations ====================
CASE iStep OF
	
	0: // Read: 16#8011:11 - Max current, Peak current [mA]
	
		// Execute read only if DriveRef is OK
		IF bDriveRefOK THEN
			fbCoERead.nIndex			:= 16#8011;
			fbCoERead.nSubIndex			:= 16#11;
			fbCoERead.pDstBuf			:= ADR(dwPeakCurrent);
			fbCoERead.cbBufLen			:= SIZEOF(dwPeakCurrent);
			fbCoERead.bExecute			:= TRUE;
			iStep 						:= iStep + 10; 
		END_IF
	
	10:	// Wait till read finish
	
		IF NOT fbCoERead.bBusy THEN
			fbCoERead.bExecute			:= FALSE;
			IF fbCoERead.bError THEN
				wInitErrorCount 		:= wInitErrorCount + 1;
				// Count > 10 then go to error and wait for reset, if not wait in warning step
				IF wInitErrorCount > 10 THEN
					uiAdsErrId			:= fbCoERead.iAdsErrId;
					uiCANopenErrId		:= fbCoERead.iCANopenErrId;
					iStep				:= 1000;								// Error step
				ELSE
					iStep				:= 900;									// Warning step
				END_IF
			ELSE
				iStep 					:= iStep + 10;
			END_IF
		END_IF
		
	20: // Read: 16#8011:12 - Rated current [mA]
	
		// Execute read only if DriveRef is OK
		IF bDriveRefOK THEN
			fbCoERead.nIndex			:= 16#8011;
			fbCoERead.nSubIndex			:= 16#12;
			fbCoERead.pDstBuf			:= ADR(dwRatedCurrent);
			fbCoERead.cbBufLen			:= SIZEOF(dwRatedCurrent);
			fbCoERead.bExecute			:= TRUE;
			iStep 						:= iStep + 10; 
		END_IF
	
	30:	// Wait till read finish
	
		IF NOT fbCoERead.bBusy THEN
			fbCoERead.bExecute			:= FALSE;
			IF fbCoERead.bError THEN
				wInitErrorCount 		:= wInitErrorCount + 1;
				// Count > 10 then go to error and wait for reset, if not wait in warning step
				IF wInitErrorCount > 10 THEN
					uiAdsErrId			:= fbCoERead.iAdsErrId;
					uiCANopenErrId		:= fbCoERead.iCANopenErrId;
					iStep				:= 1000;								// Error step
				ELSE
					iStep				:= 900;									// Warning step
				END_IF
			ELSE
				iStep 					:= iStep + 10;
			END_IF
		END_IF
		
	40: // Read: 16#8011:16 - Torque constant [mNm/A]
	
		// Execute read only if DriveRef is OK
		IF bDriveRefOK THEN
			fbCoERead.nIndex			:= 16#8011;
			fbCoERead.nSubIndex			:= 16#16;
			fbCoERead.pDstBuf			:= ADR(dwTorqueConstant);
			fbCoERead.cbBufLen			:= SIZEOF(dwTorqueConstant);
			fbCoERead.bExecute			:= TRUE;
			iStep 						:= iStep + 10; 
		END_IF
	
	50:	// Wait till read finish
	
		IF NOT fbCoERead.bBusy THEN
			fbCoERead.bExecute			:= FALSE;
			IF fbCoERead.bError THEN
				wInitErrorCount 		:= wInitErrorCount + 1;
				// Count > 10 then go to error and wait for reset, if not wait in warning step
				IF wInitErrorCount > 10 THEN
					uiAdsErrId			:= fbCoERead.iAdsErrId;
					uiCANopenErrId		:= fbCoERead.iCANopenErrId;
					iStep				:= 1000;								// Error step
				ELSE
					iStep				:= 900;									// Warning step
				END_IF
			ELSE
				iStep 					:= iStep + 10;
			END_IF
		END_IF

	60: // Read: 16#8010:54 - Feature bits
	
		// Execute read only if DriveRef is OK
		IF bDriveRefOK THEN
			fbCoERead.nIndex			:= 16#8010;
			fbCoERead.nSubIndex			:= 16#54;
			fbCoERead.pDstBuf			:= ADR(dwFeatureBits);
			fbCoERead.cbBufLen			:= SIZEOF(dwFeatureBits);
			fbCoERead.bExecute			:= TRUE;
			iStep 						:= iStep + 10; 
		END_IF
	
	70:	// Wait till read finish
	
		IF NOT fbCoERead.bBusy THEN
			fbCoERead.bExecute			:= FALSE;
			IF fbCoERead.bError THEN
				wInitErrorCount 		:= wInitErrorCount + 1;
				// Count > 10 then go to error and wait for reset, if not wait in warning step
				IF wInitErrorCount > 10 THEN
					uiAdsErrId			:= fbCoERead.iAdsErrId;
					uiCANopenErrId		:= fbCoERead.iCANopenErrId;
					iStep				:= 1000;								// Error step
				ELSE
					iStep				:= 900;									// Warning step
				END_IF
			ELSE
				iStep 					:= 100;
			END_IF
		END_IF
	
	100: // Calculate Sf
	
		bRMSValue						:= dwFeatureBits.0;											// If RMS then don't div by SQRT(2)
		rPeakCurrent 					:= DWORD_TO_REAL(dwPeakCurrent) / 1000.0;					// In [A]
		rRatedCurrent	 				:= DWORD_TO_REAL(dwRatedCurrent) / 1000.0;					// In [A]
		rSfCurrent 						:= rRatedCurrent / 100.0 / SEL(bRMSValue,SQRT(2),1 );		// iTorque -1000..1000 --> - rPeakCurrent .. rPeakCurrent [A]
		rWarningCurrent 				:= rRatedCurrent;
		rSfTorque	 					:= DWORD_TO_REAL(dwTorqueConstant) / 1000.0;				// [mNm / A]  -->  [Nm/A]
		
		iStep 							:= 200;
		
	200: // Read profile MDP 742 or DS 402:
	
			// We have to read device name Index 1008:0 - STRING
			// EL72x1-0000 --> MDP 742: A011:11 Motor I2T temperature [%] USINT
			// EL72x1-0001 --> DS 402: 2031:11 Motor I2T temperature [%] USINT
	
		// Execute read only if DriveRef is OK
		IF bDriveRefOK THEN
			fbCoERead.nIndex			:= 16#1008;
			fbCoERead.nSubIndex			:= 0;
			fbCoERead.pDstBuf			:= ADR(sDeviceName);
			fbCoERead.cbBufLen			:= SIZEOF(sDeviceName);
			fbCoERead.bExecute			:= TRUE;
			iStep 						:= iStep + 10; 
		END_IF
	
	210:	// Wait till read finish
	
		IF NOT fbCoERead.bBusy THEN
			fbCoERead.bExecute			:= FALSE;
			IF fbCoERead.bError THEN
				wInitErrorCount 		:= wInitErrorCount + 1;
				// Count > 10 then go to error and wait for reset, if not wait in warning step
				IF wInitErrorCount > 10 THEN
					uiAdsErrId			:= fbCoERead.iAdsErrId;
					uiCANopenErrId		:= fbCoERead.iCANopenErrId;
					iStep				:= 1000;								// Error step
				ELSE
					iStep				:= 900;									// Warning step
				END_IF
			ELSE
				iStep 					:= iStep + 10;
			END_IF
		END_IF

	220: // Check last digit in device name 0 - MDP742, 1 - DS402
	
	sNo 								:=  MID(sDeviceName, 1, FIND(sDeviceName, '-') + 4);
	bMDP742Profile 						:= 	sNo = '0';
	bDS402Profile 						:= 	sNo = '1';
	bMDP742Profile 						:= 	sNo = '4';
	// If 0 or 1 then go to next step, if other No - not implemented yet
	IF bMDP742Profile OR bDS402Profile THEN
		wMotorI2TIndex					:= SEL(bMDP742Profile, 16#2031, 16#A011);
		iStep 							:= iStep + 10;
	ELSE
		iStep							:= 1000;					// Error step
	END_IF

	230: // Read profile MDP 742 or DS 402:
	
			// EL72x1-0000 --> MDP 742: A011:11 Motor I2T temperature [%] USINT
			// EL72x1-0001 --> DS 402: 2031:11 Motor I2T temperature [%] USINT
	
		// Execute read only if DriveRef is OK and read trigger
		fbCoERead.nIndex				:= wMotorI2TIndex;
		fbCoERead.nSubIndex				:= 16#11;
		fbCoERead.pDstBuf				:= ADR(usiI2T);
		fbCoERead.cbBufLen				:= SIZEOF(usiI2T);
		fbCoERead.bExecute				:= bDriveRefOK AND tonWait.Q;
		IF fbCoERead.bBusy THEN
			iStep 						:= iStep + 10;
		END_IF
	
	240:	// Wait till read finish
	
		IF NOT fbCoERead.bBusy THEN
			fbCoERead.bExecute			:= FALSE;
			IF fbCoERead.bError THEN
				wInitErrorCount 		:= wInitErrorCount + 1;
				// Count > 10 then go to error and wait for reset, if not wait in warning step
				IF wInitErrorCount > 10 THEN
					uiAdsErrId			:= fbCoERead.iAdsErrId;
					uiCANopenErrId		:= fbCoERead.iCANopenErrId;
					iStep				:= 1000;								// Error step
				ELSE
					iStep				:= 900;									// Warning step
				END_IF
			ELSE
				rI2T					:= USINT_TO_REAL(usiI2T);				// Konwersja i przepisanie
				iStep 					:= iStep - 10;
			END_IF
		END_IF
	
	900: // Warning - wait and repeat read - problem during read motor data, i.e. EtherCAT doesn't work yet
		IF tonWait.Q THEN
			iStep 						:= 0;	// Repeat initialization phase 
		END_IF
			  
			  
	1000: // Error - wait for reset 
		;
END_CASE
//===============================================================

bError		 							:= iStep = 1000;
bInitialized 							:= iStep >= 230 AND NOT bError;
ACT_Calculations();

//======================== Save I2T max value ======================
IF rI2TMax < rI2T THEN
	rI2TMax 							:= rI2T;
END_IF

//========================= Warning =============================
bWarning								:= rCurrentF > rWarningCurrent;

//===================== Limit output torque =====================
IF rTorqueLimit < rTorqueLimitLow THEN
	uiBipolarTorqueLimitValue 			:= REAL_TO_UINT(rTorqueLimitHigh);			// Secure against 0 value - probably empty var connected to input
ELSE
	uiBipolarTorqueLimitValue 			:= REAL_TO_UINT(LIMIT(rTorqueLimitLow,rTorqueLimit,rTorqueLimitHigh)) * 10;
END_IF
//====================== Call CoE read FB =======================
fbCoERead(stDriveRef:= stDriveRef);

ACTION ACT_Calculations:
//============== Raw values - always avaliable ==================
rTorquePerc								:= LREAL_TO_REAL(Axis.NcToPlc.ActTorque); 		// [%]
rTorqueRAW 								:= rTorquePerc * 10;							// -1000 .. 1000 - RAW values the same as process image
//===================== Filter current value ====================
fbFilterEx(rIn:= rTorqueRAW, tTimeConstant:= T#1S);

// Calculations	- possible only with params
IF bInitialized THEN
	rCurrent 							:= rTorqueRAW * rSfCurrent;
	rTorque 							:= rCurrent * rSfTorque;

	
	rCurrentF 							:= fbFilterEx.rOut * rSfCurrent;
	rTorqueF 							:= (fbFilterEx.rOut * rSfTorque) / 100;
END_IF

//=============== Save torque and current max values ===============
IF ABS(rCurrentMax) < ABS(rCurrentF) THEN
	rTorquePercMax						:= rTorquePerc;
	rCurrentMax 						:= rCurrentF;
	rTorqueMax 							:= rTorqueF;
END_IF
END_ACTION

ACTION ACT_Init_Reset:
//============== Reset max values and FB ========================
rtReset(CLK:= bReset);
IF rtReset.Q THEN
	fbCoERead.bExecute					:= FALSE;
	// FB Outputs
	rWarningCurrent						:= 0;
	rTorquePerc							:= 0;
	rTorquePercMax						:= 0;
	rTorque								:= 0;
	rTorqueF							:= 0;
	rTorqueMax							:= 0;
	rCurrent							:= 0;
	rCurrentF							:= 0;
	rCurrentMax							:= 0;
	rI2T								:= 0;
	rI2TMax								:= 0;
	uiAdsErrId		 					:= 0;
	uiCANopenErrId	 					:= 0;
	// Internal
	iStep								:= 0;
	wInitErrorCount						:= 0;
	rTorqueRAW							:= 0;
	rSfTorque							:= 0;
	rSfCurrent							:= 0;
	wInitErrorCount						:= 0;
	rPeakCurrent						:= 0;
	rRatedCurrent						:= 0;
	bRMSValue							:= FALSE;
	dwPeakCurrent						:= 0;
	dwRatedCurrent						:= 0;
	dwTorqueConstant					:= 0;
	dwFeatureBits						:= 0;
	sDeviceName							:= '';
	sNo									:= '';
	usiI2T								:= 0;
	bDS402Profile						:= FALSE;
	bMDP742Profile						:= FALSE;
	wMotorI2TIndex						:= 0;
END_IF
END_ACTION

END_FUNCTION_BLOCK

// ---- AxisOnline/POUs/EL72xx/FB_HoldingBrakeCtrlEL72xx.TcPOU
//==================================================================================================
//							Beckhoff Automation Poland
//									11.07.2018
//	Blok funkcyjny kontroli luzownika w silniku podpietym do EL72xx. Mozliwy jest jedynie force unlock.
//	Dzialania na obiekcie:	: 8012:01 (MDP742) lub 2004:01 (DS402)
//
//  v1.0	|| TC v 3.1.4022.22		|| - pierwsza wersja
//==================================================================================================
FUNCTION_BLOCK FB_HoldingBrakeCtrlEL72xx
VAR_INPUT
	bForceUnlock					: BOOL;								// Rising/falling edhe executes CMD: Manual override (release) of the motor holding brake 
																		// and reset - if there is error - falling edge reinits FB
	stDriveRef						: ST_DriveRef;
END_VAR
VAR_OUTPUT
	bBusy							: BOOL;
	bError							: BOOL; 							// General error: parameter or CoE read.
	uiAdsErrId						: UINT;								// Forwarded output FB_CoERead_ByDriveRef
	uiCANopenErrId					: UINT;								// Forwarded output FB_CoERead_ByDriveRef
END_VAR
VAR
	//======================= Internal var ===========================
	iStep							: INT;								// Case instruction	
	wInitErrorCount					: WORD;								// Initialization error counter, if bigger then 10 then error
	wManualOverrideIndex			: WORD;								// Manual override (release) of the motor holding brake:
																		// MDP742: 8012:01
																		// DS402: 2004:01
	bDriveRefOK						: BOOL;								// stDriveRef contains necessary data to read CoE
	bExecute						: BOOL;
	bDS402Profile					: BOOL;								// Flag DS402
	bMDP742Profile					: BOOL;								// Flag MDP742	
	bInitialized					: BOOL;
	sDeviceName						: STRING;							// 
	sNo								: STRING(1);						// xxxxxxx-000Y - char Y	
	//=========================== FBs ================================																
	rtForceUnlock					: R_TRIG;
	ftForceUnlock					: F_TRIG;
	tonWait							: TON;								// Wait timer
	fbCoERead						: FB_CoERead_ByDriveRef;			// FB for read CoE parameters
	fbForceUnlock					: FB_CoEWrite_ByDriveRef;
END_VAR

//=================== Call triggers and timers ==================
tonWait(IN:= NOT tonWait.Q, PT:= T#1S);
rtForceUnlock(CLK:= bForceUnlock);
ftForceUnlock(CLK:= bForceUnlock);

//======= Check for parameter error - each cycle ================
bDriveRefOK 							:= (stDriveRef.nSlaveAddr <> 0) AND (stDriveRef.sNetId <> '');

//============= Read params and calculations ====================
CASE iStep OF
	
	0: // Read profile MDP 742 or DS 402:
	
			// We have to read device name Index 1008:0 - STRING
			// EL72x1-0000 --> MDP 742:
			// EL72x1-0001 --> DS 402:
	
		// Execute read only if DriveRef is OK
		IF bDriveRefOK THEN
			fbCoERead.nIndex			:= 16#1008;
			fbCoERead.nSubIndex			:= 0;
			fbCoERead.pDstBuf			:= ADR(sDeviceName);
			fbCoERead.cbBufLen			:= SIZEOF(sDeviceName);
			fbCoERead.bExecute			:= TRUE;
			iStep 						:= iStep + 10; 
		END_IF
	
	10:	// Wait till read finish
	
		IF NOT fbCoERead.bBusy THEN
			fbCoERead.bExecute			:= FALSE;
			IF fbCoERead.bError THEN
				wInitErrorCount 		:= wInitErrorCount + 1;
				// Count > 10 then go to error and wait for reset, if not wait in warning step
				IF wInitErrorCount > 10 THEN
					uiAdsErrId			:= fbCoERead.iAdsErrId;
					uiCANopenErrId		:= fbCoERead.iCANopenErrId;
					iStep				:= 1000;								// Error step
				ELSE
					iStep				:= 900;									// Warning step
				END_IF
			ELSE
				iStep 					:= iStep + 10;
			END_IF
		END_IF

	20: // Check last digit in device name 0 - MDP742, 1 - DS402
	
	sNo 								:=  MID(sDeviceName, 1, FIND(sDeviceName, '-') + 4);
	bMDP742Profile 						:= 	sNo = '0';
	bDS402Profile 						:= 	sNo = '1';
	// If 0 or 1 then go to next step, if other No - not implemented yet
	IF bMDP742Profile OR bDS402Profile THEN
		wManualOverrideIndex			:= SEL(bMDP742Profile, 16#2004, 16#8012);
		iStep 							:= 100;
	ELSE
		iStep							:= 1000;					// Error step
	END_IF
	
	100: // Initialized - holding brake control possible
		fbForceUnlock.bExecute			:= rtForceUnlock.Q OR ftForceUnlock.Q;
		IF fbForceUnlock.bBusy THEN
			iStep 						:= iStep + 10;
		END_IF

	110: // Wait till write finish
	
		IF NOT fbForceUnlock.bBusy THEN
			fbForceUnlock.bExecute		:= FALSE;
			IF fbForceUnlock.bError THEN
				uiAdsErrId				:= fbForceUnlock.iAdsErrId;
				uiCANopenErrId			:= fbForceUnlock.iCANopenErrId;
			ELSE
				iStep 					:= iStep - 10;
			END_IF
		END_IF
	
	900: // Warning - wait and repeat read - problem during read motor data, i.e. EtherCAT doesn't work yet
		IF tonWait.Q THEN
			iStep 						:= 0;	// Repeat initialization phase 
		END_IF
			  
	1000: // Error - wait for reset 
		IF ftForceUnlock.Q THEN
			uiAdsErrId					:= 0;
			uiCANopenErrId				:= 0;
			wInitErrorCount				:= 0;
			wManualOverrideIndex		:= 0;
			sDeviceName					:= '';
			sNo							:= '';
			bDS402Profile				:= FALSE;
			bMDP742Profile				:= FALSE;
			iStep						:= 0;
		END_IF
END_CASE
//===============================================================

bError		 							:= iStep = 1000;
bInitialized 							:= iStep >= 100 AND iStep < 900;

//================== Call CoE read/write FB =====================
fbCoERead(stDriveRef:= stDriveRef);

fbForceUnlock	(	stDriveRef				:= stDriveRef, 
					nIndex					:= wManualOverrideIndex, 
					nSubIndex				:= 16#01, 
					pSrcBuf					:= ADR(bForceUnlock), 
					cbBufLen				:= SIZEOF(bForceUnlock));
//===============================================================

END_FUNCTION_BLOCK

// ---- AxisOnline/POUs/EL72xx/FB_ReadChannelErrorCodeEL72xx.TcPOU
//==================================================================================================
//							Beckhoff Automation Poland
//									11.07.2018
//	This object shall provide the text id of the last DiagMessage of type error, which occurred in this axis.
//  v1.0	|| TC v 3.1.4022.22		|| - pierwsza wersja
//==================================================================================================
FUNCTION_BLOCK FB_ReadChannelErrorCodeEL72xx
VAR_INPUT
	bExecute 						: BOOL;
	stDriveRef						: ST_DriveRef;						// 
END_VAR
VAR_OUTPUT
	bBusy							: BOOL;
	bError							: BOOL; 							// General error: parameter or CoE read.
	uiAdsErrId						: UINT;								// Forwarded output FB_CoERead_ByDriveRef
	uiCANopenErrId					: UINT;								// Forwarded output FB_CoERead_ByDriveRef
	uiChannelErrorCode				: UINT;								// Error Code: 16#10F3: usiSubindexOfLatestMessage
	{attribute 'displaymode':='hex'}
	uiChannelErrorCodeHex			: UINT;								// Error Code: 16#10F3: usiSubindexOfLatestMessage
END_VAR
VAR
	fbCoERead						: FB_CoERead_ByDriveRef;			// FB for read CoE parameters
	bDriveRefOK						: BOOL;
	usiSubindexOfLatestMessage		: USINT;
	arrMessage						: ARRAY [1..28] OF BYTE;
	iStep							: INT;
	rtExecute						: R_TRIG;
END_VAR

//=================== Call triggers and timers ==================
rtExecute(CLK:= bExecute, Q=> );
IF rtExecute.Q THEN
	iStep	:= 0;
END_IF

//======= Check for parameter error - each cycle ================
bDriveRefOK 							:= (stDriveRef.nSlaveAddr <> 0) AND (stDriveRef.sNetId <> '');

//======================== Read params ==========================
CASE iStep OF
	
	0, 1000: // Read: 16#10F3:02 - Newest Message, Subindex of the latest message: UINT8

		// Execute read only if DriveRef is OK
		IF bDriveRefOK AND rtExecute.Q THEN
			fbCoERead.nIndex			:= 16#10F3;
			fbCoERead.nSubIndex			:= 16#02;
			fbCoERead.pDstBuf			:= ADR(usiSubindexOfLatestMessage);
			fbCoERead.cbBufLen			:= SIZEOF(usiSubindexOfLatestMessage);
			fbCoERead.bExecute			:= TRUE;
			iStep 						:= 10;
		END_IF
	
	10:	// Wait till read finish
	
		IF NOT fbCoERead.bBusy THEN
			fbCoERead.bExecute			:= FALSE;
			IF fbCoERead.bError THEN
				uiAdsErrId				:= fbCoERead.iAdsErrId;
				uiCANopenErrId			:= fbCoERead.iCANopenErrId;
				iStep					:= 1000;								// Error step
			ELSE
				iStep 					:= iStep + 10;
			END_IF
		END_IF
		
	20: // Read: 16#10F3:usiSubindexOfLatestMessage - Message usiSubindexOfLatestMessage-5
	
		// Execute read only if DriveRef is OK
		IF bDriveRefOK THEN
			fbCoERead.nIndex			:= 16#10F3;
			fbCoERead.nSubIndex			:= usiSubindexOfLatestMessage;
			fbCoERead.pDstBuf			:= ADR(arrMessage);
			fbCoERead.cbBufLen			:= SIZEOF(arrMessage);
			fbCoERead.bExecute			:= TRUE;
			iStep 						:= iStep + 10; 
		END_IF
	
	30:	// Wait till read finish

		IF NOT fbCoERead.bBusy THEN
			fbCoERead.bExecute			:= FALSE;
			IF fbCoERead.bError THEN
				uiAdsErrId				:= fbCoERead.iAdsErrId;
				uiCANopenErrId			:= fbCoERead.iCANopenErrId;
				iStep					:= 1000;								// Error step
			ELSE
				uiChannelErrorCode		:= 16#0100 * arrMessage[8] + arrMessage[7];
				iStep 					:= 0;									// Read Done
			END_IF
		END_IF

END_CASE

bError									:= iStep = 1000;
bBusy									:= iStep <> 0 AND NOT bError;
//====================== Call CoE read FB =======================
fbCoERead(stDriveRef:= stDriveRef);

uiChannelErrorCodeHex					:= uiChannelErrorCode;

END_FUNCTION_BLOCK

// ---- AxisOnline/POUs/AX5xxx/FB_HoldingBrakeCtrlAX5000.TcPOU
//==================================================================================================
//							Beckhoff Automation Poland
//									23.05.2018
//	Blok funkcyjny kontroli luzownika w silniku podpietym do AX5000. Przewaga ForceLock
//	Datatype:		ENUM (INT16)
//	Enum Value:		0 (0x00): 	Release_force
//					1 (0x01): 	Force_lock
//					2 (0x02): 	Force_unlock
//
// 	v1.1	|| TC v 3.1.4022.16	|| - optymalizacja kodu
//  v1.0	|| TC v 3.1.4022.16	|| - pierwsza wersja
//==================================================================================================
FUNCTION_BLOCK FB_HoldingBrakeCtrlAX5000
VAR_INPUT
	bForceLock 						: BOOL;								// 
	bForceUnlock					: BOOL;								// 
END_VAR
VAR_OUTPUT
	bBusy							: BOOL;
	bError							: BOOL; 							// General error: parameter or CoE read.
																		// If bError = TRUE and bInitialized = FALSE - error during read motor data.
																		// If bError = TRUE and bInitialized = TRUE and (iAdsErrId <> 0 or iCANopenErrId <> 0) then I2T read error
																		// If bError = TRUE and bInitialized = TRUE and iAdsErrId = 0 and iCANopenErrId = 0 then parameter error: rTorqueLimit outside permitted range rTorqueLimitLow..rTorqueLimitHigh or Empty stDriveRef
	iAdsErrId						: UINT;								// Forwarded output FB_SoEWrite
	iSecErrId						: UINT;								// Forwarded output FB_SoEWrite
END_VAR
VAR_IN_OUT
	Axis							: AXIS_REF;
END_VAR
VAR
	bExecute						: BOOL;
	iMotorBrakeForce				: INT;								// 0 - Release_force, 1 - Force_lock, 2 - Force_unlock
	fbSoEWrite						: FB_SoEWrite;
	rtForceLock						: R_TRIG;
	rtForceUnlock					: R_TRIG;
	ftForceLock						: F_TRIG;
	ftForceUnlock					: F_TRIG;
END_VAR

{region "Call triggers"}
//======================= Call triggers =========================
rtForceLock(CLK:= bForceLock);
ftForceLock(CLK:= bForceLock);
rtForceUnlock(CLK:= bForceUnlock);
ftForceUnlock(CLK:= bForceUnlock);
bExecute								:= rtForceLock.Q OR ftForceLock.Q OR rtForceUnlock.Q OR ftForceUnlock.Q;
//===============================================================
{endregion}
{region "Main code"}
//========================= Main code ===========================
IF bExecute THEN
	iMotorBrakeForce 						:= 0;										// Clear value
	iMotorBrakeForce.1 						:= bForceUnlock;							// Set force unlock bit
	iMotorBrakeForce 						:= SEL(bForceLock, iMotorBrakeForce, 1);	// Set force lock bit, it has higher priority than unlock
END_IF
	 
fbSoEWrite(
	NetId			:= '' , 
	Idn				:= P_0_IDN + 96 , 
	Element			:= 16#40 , 
	pSrcBuf			:= ADR(iMotorBrakeForce), 
	BufLen			:= SIZEOF(iMotorBrakeForce) , 
	Execute			:= bExecute , 
	Timeout			:= T#2S, 
	Axis			:= Axis , 
	Busy			=> bBusy , 
	Error			=> bError, 
	AdsErrId		=> iAdsErrId, 
	SercosErrId		=> iSecErrId );
//===============================================================
{endregion}

END_FUNCTION_BLOCK

// ---- AxisOnline/POUs/AX5xxx/F_AX5xErrMsg.TcPOU
//==================================================================================================
//							Beckhoff Automation Poland
//								7.12.2018
//		Funkcja konwertujaca nr bledu na opis
// 	v1.0	|| TC v 3.1.4022.27	|| - pierwsza wersja
//==================================================================================================
FUNCTION F_AX5xErrMsg : STRING(255)
VAR_INPUT
	uiDriveError : UINT;
END_VAR

IF uiDriveError < 1 THEN
	F_AX5xErrMsg := '';
	RETURN;
END_IF

